Staubli VAL3: powerOn.pgx

program powerOn()
begin
 enablePower()
 if (watch(isPowered(),5)==false)
  putln("Arm power supply cannot be switched on")
 endIf
 message="enablePower:done"
 taskCreate "sendStatus",100,sendStatus()
 taskKill ("powerOn")
end
